# B&R Automation Studio project Ampel (part 6)

```cpp
	processRequest();
}

template <typename TG_, typename TA_>
HFSM2_CONSTEXPR(14)
void
R_<TG_, TA_>::immediateRestart(const StateID stateId_) noexcept {
	restart(stateId_);

	processRequest();
}

template <typename TG_, typename TA_>
HFSM2_CONSTEXPR(14)
void
R_<TG_, TA_>::immediateResume(const StateID stateId_) noexcept {
	resume(stateId_);

	processRequest();
}

template <typename TG_, typename TA_>
HFSM2_CONSTEXPR(14)
void
R_<TG_, TA_>::immediateSelect(const StateID stateId_) noexcept {
	select(stateId_);

	processRequest();
}

#if HFSM2_UTILITY_THEORY_AVAILABLE()

template <typename TG_, typename TA_>
HFSM2_CONSTEXPR(14)
void
R_<TG_, TA_>::immediateUtilize(const StateID stateId_) noexcept {
	utilize(stateId_);

	processRequest();
}

template <typename TG_, typename TA_>
HFSM2_CONSTEXPR(14)
void
R_<TG_, TA_>::immediateRandomize(const StateID stateId_) noexcept {
	randomize(stateId_);

	processRequest();
}

#endif

template <typename TG_, typename TA_>
HFSM2_CONSTEXPR(14)
void
R_<TG_, TA_>::reset() noexcept {
	HFSM2_ASSERT(_core.registry.isActive());

TransitionSets currentTransitions;
PlanControl control{_core, currentTransitions};

	_apex.deepExit(control);

	HFSM2_IF_TRANSITION_HISTORY(_core.transitionTargets.clear());
	HFSM2_IF_TRANSITION_HISTORY(_core.previousTransitions.clear());

	_core.registry.clear();
	// TODO: clear _core.requests
	// TODO: clear _core.rng			// HFSM2_IF_UTILITY_THEORY()
	// TODO: clear _core.planData		// HFSM2_IF_PLANS()
	// TODO: clear _activityHistory		// HFSM2_IF_STRUCTURE_REPORT()

_apex.deepRequestChange(control, {TransitionType::RESTART, INVALID_SHORT});
	_apex.deepEnter(control);
}

#if HFSM2_TRANSITION_HISTORY_AVAILABLE()

template <typename TG_, typename TA_>
HFSM2_CONSTEXPR(14)
bool
R_<TG_, TA_>::replayTransitions(const Transition* const transitions,
							  const Short count) noexcept
{
	HFSM2_ASSERT(transitions);
	HFSM2_ASSERT(_core.registry.isActive());

	_core.transitionTargets  .clear();
	_core.previousTransitions.clear();

	if (HFSM2_CHECKED(transitions && count)) {
TransitionSets currentTransitions;
PlanControl control{_core, currentTransitions};

		if (HFSM2_CHECKED(applyRequests(control, transitions, count))) {
for (Short i = 0; i < count; ++i)
				_core.previousTransitions.emplace(transitions[i]);

			_apex.deepChangeToRequested(control);

			_core.registry.clearRequests();

			HFSM2_IF_ASSERT(HFSM2_IF_PLANS(_core.planData.verifyPlans()));
			HFSM2_IF_STRUCTURE_REPORT(udpateActivity());

			return true;
		}
	}

	return false;
}

template <typename TG_, typename TA_>
template <Long NCount>
HFSM2_CONSTEXPR(14)
bool
R_<TG_, TA_>::replayTransitions(const DynamicArrayT<Transition, NCount>& transitions) noexcept {
	if (transitions.count())
		return replayTransitions(&transitions[0],
								 transitions.count());
	else
		return false;
}

template <typename TG_, typename TA_>
HFSM2_CONSTEXPR(14)
const typename R_<TG_, TA_>::Transition*
R_<TG_, TA_>::lastTransitionTo(const StateID stateId_) const noexcept {
	HFSM2_ASSERT(_core.registry.isActive());

	if (HFSM2_CHECKED(stateId_ < StateList::SIZE)) {
		const Short index = _core.transitionTargets[stateId_];

		if (index < _core.previousTransitions.count())
			return &_core.previousTransitions[index];
	}

	return nullptr;
}

#endif

template <typename TG_, typename TA_>
HFSM2_CONSTEXPR(14)
void
R_<TG_, TA_>::initialEnter() noexcept {
	HFSM2_ASSERT(!_core.registry.isActive());
	HFSM2_ASSERT(_core.requests.count() == 0);
	HFSM2_IF_TRANSITION_HISTORY(_core.transitionTargets.clear());
	HFSM2_IF_TRANSITION_HISTORY(HFSM2_ASSERT(_core.previousTransitions.count() == 0));

TransitionSets currentTransitions;
TransitionSet  pendingTransitions;

RegistryBackUp undo;
PlanControl control{_core, currentTransitions};

_apex.deepRequestChange(control, {TransitionType::RESTART, INVALID_SHORT});

	cancelledByEntryGuards(currentTransitions,
						   pendingTransitions);

for (Long i = 0;
		 i < SUBSTITUTION_LIMIT && _core.requests.count();
		 ++i)
	{
		backup(_core.registry, undo);

		if (applyRequests(currentTransitions,
						  control))
		{
pendingTransitions = _core.requests;
			_core.requests.clear();

			if (cancelledByEntryGuards(currentTransitions,
									   pendingTransitions))
			{
				HFSM2_BREAK();

				restore(_core.registry, undo);
			} else
currentTransitions += pendingTransitions;

			pendingTransitions.clear();
		} else
			_core.requests.clear();
	}
	HFSM2_ASSERT(_core.requests.count() == 0);
	HFSM2_IF_TRANSITION_HISTORY(_core.previousTransitions = currentTransitions);

	_apex.deepEnter(control);

	_core.registry.clearRequests();

	HFSM2_IF_ASSERT(HFSM2_IF_PLANS(_core.planData.verifyPlans()));
	HFSM2_IF_STRUCTURE_REPORT(udpateActivity());
}

template <typename TG_, typename TA_>
HFSM2_CONSTEXPR(14)
void
R_<TG_, TA_>::finalExit() noexcept {
	HFSM2_ASSERT(_core.registry.isActive());

TransitionSets emptyTransitions;
PlanControl control{_core, emptyTransitions};

	_apex.deepExit(control);

	_core.registry.clear();
	_core.requests.clear();

#if HFSM2_PLANS_AVAILABLE()
	_core.planData.clear();
#endif

#if HFSM2_UTILITY_THEORY_AVAILABLE()
	// TODO: _core.rng.clear();
#endif

#if HFSM2_TRANSITION_HISTORY_AVAILABLE()
	_core.transitionTargets  .clear();
	_core.previousTransitions.clear();
#endif

	HFSM2_IF_STRUCTURE_REPORT(udpateActivity());
}

template <typename TG_, typename TA_>
HFSM2_CONSTEXPR(14)
void
R_<TG_, TA_>::processRequest() noexcept {
	HFSM2_IF_ASSERT(HFSM2_IF_PLANS(_core.planData.verifyPlans()));

TransitionSets currentTransitions;
	HFSM2_IF_TRANSITION_HISTORY(_core.transitionTargets.clear());

	if (_core.requests.count()) {
		processTransitions(currentTransitions);

		HFSM2_IF_ASSERT(HFSM2_IF_PLANS(_core.planData.verifyPlans()));
		HFSM2_IF_STRUCTURE_REPORT(udpateActivity());
	}

	HFSM2_IF_TRANSITION_HISTORY(_core.previousTransitions = currentTransitions);
}

template <typename TG_, typename TA_>
HFSM2_CONSTEXPR(14)
void
R_<TG_, TA_>::processTransitions(TransitionSets& currentTransitions) noexcept {
	HFSM2_ASSERT(_core.registry.isActive());
	HFSM2_ASSERT(_core.requests.count());

TransitionSet pendingTransitions;

RegistryBackUp registryUndo;
PlanControl control{_core, currentTransitions};

for (Long i = 0;
		 i < SUBSTITUTION_LIMIT && _core.requests.count();
		 ++i)
	{
		backup(_core.registry, registryUndo);

		if (applyRequests(currentTransitions,
						  control))
		{
pendingTransitions = _core.requests;
			_core.requests.clear();

			if (cancelledByGuards(currentTransitions,
								  pendingTransitions))
			{
				HFSM2_IF_TRANSITION_HISTORY(_core.transitionTargets.clear());
				restore(_core.registry, registryUndo);
			} else
currentTransitions += pendingTransitions;

			pendingTransitions.clear();
		} else
			_core.requests.clear();
	}
	HFSM2_ASSERT(_core.requests.count() == 0);

	if (currentTransitions.count())
		_apex.deepChangeToRequested(control);

	_core.registry.clearRequests();
}

template <typename TG_, typename TA_>
HFSM2_CONSTEXPR(14)
bool
R_<TG_, TA_>::applyRequests(const TransitionSets& currentTransitions,
							Control& control) noexcept
{
bool changesMade = false;

for (Short i = 0; i < _core.requests.count(); ++i)
		changesMade |= applyRequest(currentTransitions, control, _core.requests[i], i);

return changesMade;
}

template <typename TG_, typename TA_>
HFSM2_CONSTEXPR(14)
bool
R_<TG_, TA_>::applyRequest(const TransitionSets& currentTransitions,
						   Control& control,
						   const Transition& request,
						   const Short index) noexcept
{
for (Short i = 0; i < currentTransitions.count(); ++i)
if (currentTransitions[i] == request)
			return false;

	switch (request.type) {
	case TransitionType::CHANGE:
	case TransitionType::RESTART:
	case TransitionType::RESUME:
	case TransitionType::SELECT:

#if HFSM2_UTILITY_THEORY_AVAILABLE()
	case TransitionType::UTILIZE:
	case TransitionType::RANDOMIZE:
#endif

		// TODO: have both return success status
		if (_core.registry.requestImmediate(request))
_apex.deepForwardActive(control, {request.type, index});
		else
_apex.deepRequest	   (control, {request.type, index});

		return true;

	case TransitionType::SCHEDULE:
		_core.registry.requestScheduled(request.destination);

		return false;

	default:
		HFSM2_BREAK();

		return false;
	}
}

template <typename TG_, typename TA_>
HFSM2_CONSTEXPR(14)
bool
R_<TG_, TA_>::cancelledByEntryGuards(const TransitionSets& currentTransitions,
									 const TransitionSet&  pendingTransitions) noexcept
{
GuardControl guardControl{_core,
							  currentTransitions,
							  pendingTransitions};

	return _apex.deepEntryGuard(guardControl);
}

template <typename TG_, typename TA_>
HFSM2_CONSTEXPR(14)
bool
R_<TG_, TA_>::cancelledByGuards(const TransitionSets& currentTransitions,
								const TransitionSet&  pendingTransitions) noexcept
{
GuardControl guardControl{_core,
							  currentTransitions,
							  pendingTransitions};

	return _apex.deepForwardExitGuard(guardControl) ||
		   _apex.deepForwardEntryGuard(guardControl);
}

#if HFSM2_SERIALIZATION_AVAILABLE()

template <typename TG_, typename TA_>
HFSM2_CONSTEXPR(14)
void
R_<TG_, TA_>::save(WriteStream& stream) const noexcept {
	HFSM2_ASSERT(_core.registry.isActive());

	_apex.deepSaveActive(_core.registry, stream);

	// TODO: save(stream, _core.requests);

#if HFSM2_PLANS_AVAILABLE()
	// TODO: save(stream, _core.planData);
#endif

#if HFSM2_UTILITY_THEORY_AVAILABLE()
	// TODO: save(stream, _core.rng);
#endif

#if HFSM2_TRANSITION_HISTORY_AVAILABLE()
	// TODO: save(stream, _core.transitionTargets);
	// TODO: save(stream, _core.previousTransitions);
#endif

#if HFSM2_STRUCTURE_REPORT_AVAILABLE()
	// TODO: save(stream, _activityHistory);
#endif
}

template <typename TG_, typename TA_>
HFSM2_CONSTEXPR(14)
void
R_<TG_, TA_>::load(ReadStream& stream) noexcept {
	HFSM2_ASSERT(_core.registry.isActive());

	_core.registry.clearRequests();
	_core.registry.compoResumable.clear();
	_apex.deepLoadRequested(_core.registry, stream);

	_core.requests.clear();
	// TODO: load(stream, _core.requests);

#if HFSM2_PLANS_AVAILABLE()
	_core.planData.clear();
	// TODO: load(stream, _core.planData);
#endif

#if HFSM2_UTILITY_THEORY_AVAILABLE()
	// TODO: load(stream, _core.rng);
#endif

#if HFSM2_TRANSITION_HISTORY_AVAILABLE()
	_core.transitionTargets  .clear();
	_core.previousTransitions.clear();
#endif

#if HFSM2_STRUCTURE_REPORT_AVAILABLE()
	// TODO: load(stream, _activityHistory);
#endif

TransitionSets emptyTransitions;
PlanControl control{_core, emptyTransitions};

	_apex.deepChangeToRequested(control);

	HFSM2_IF_STRUCTURE_REPORT(udpateActivity());
}

#endif

#if HFSM2_TRANSITION_HISTORY_AVAILABLE()

template <typename TG_, typename TA_>
HFSM2_CONSTEXPR(14)
bool
R_<TG_, TA_>::applyRequests(Control& control,
							const Transition* const transitions,
							const Short count) noexcept
{
TransitionSets currentTransitions;

	if (HFSM2_CHECKED(transitions && count)) {
bool changesMade = false;

for (Short i = 0; i < count; ++i)
			changesMade |= applyRequest(currentTransitions, control, transitions[i], i);

return changesMade;
	} else
		return false;
}

#endif

#if HFSM2_STRUCTURE_REPORT_AVAILABLE()

template <typename TG_, typename TA_>
HFSM2_CONSTEXPR(14)
void
R_<TG_, TA_>::getStateNames() noexcept {
StructureStateInfos stateInfos;
	_apex.deepGetNames(static_cast<Long>(-1), RegionType::COMPOSITE, 0, stateInfos);

Long margin = static_cast<Long>(-1);
for (Long s = 0; s < stateInfos.count(); ++s) {
const StructureStateInfo& stateInfo = stateInfos[s];
Prefix& prefix = _prefixes[s];

if (stateInfo.name[0] != '\0')
			_namedStates.set(s);

if (margin > stateInfo.depth && stateInfo.name[0] != '\0')
margin = stateInfo.depth;

		if (stateInfo.depth == 0)
prefix[0] = L'\0';
		else {
const Long mark = stateInfo.depth * 2 - 1;

prefix[mark + 0] = stateInfo.regionType == RegionType::COMPOSITE ? L'+' : L'+';
prefix[mark + 1] = L' ';
prefix[mark + 2] = L'\0';

for (Long d = mark; d > 0; --d)
prefix[d - 1] = L' ';

for (Long r = s; r > stateInfo.parent; --r) {
Prefix& prefixAbove = _prefixes[r - 1];

switch (prefixAbove[mark]) {
				case L' ':
prefixAbove[mark] = stateInfo.regionType == RegionType::COMPOSITE ? L'¦' : L'¦';
					break;
				case L'+':
prefixAbove[mark] = L'+';
					break;
				case L'+':
prefixAbove[mark] = L'¦';
					break;
				}
			}
		}
	}
	if (margin > 0)
		margin -= 1;

	_structure.clear();
for (Long s = 0; s < stateInfos.count(); ++s) {
const StructureStateInfo& stateInfo = stateInfos[s];
Prefix& prefix = _prefixes[s];
const Long space = stateInfo.depth * 2;

if (stateInfo.name[0] != L'\0') {
_structure.emplace(StructureEntry{false, &prefix[margin * 2], stateInfo.name});
			_activityHistory.emplace(static_cast<int8_t>(0));
		} else if (s + 1 < stateInfos.count()) {
Prefix& nextPrefix = _prefixes[s + 1];

			if (s > 0)
for (Long c = 0; c <= space; ++c)
nextPrefix[c] = prefix[c];

const Long mark = space + 1;

switch (nextPrefix[mark]) {
			case L'+':
nextPrefix[mark] = stateInfo.depth == margin ? L'+' : L'-';
				break;
			case L'¦':
nextPrefix[mark] = stateInfo.depth == margin ? L'+' : L'-';
				break;
			}
		}
	}
}

template <typename TG_, typename TA_>
HFSM2_CONSTEXPR(14)
void
R_<TG_, TA_>::udpateActivity() noexcept {
for (Long s = 0, i = 0; s < STATE_COUNT; ++s)
		if (_namedStates.get(s)) {
_structure[i].isActive = isActive(s);

typename ActivityHistory::Item& activity = _activityHistory[i];

if (_structure[i].isActive) {
				if (activity < 0)
activity = +1;
				else
activity = activity < INT8_MAX ? activity + 1 : activity;
			} else {
				if (activity > 0)
activity = -1;
				else
activity = activity > INT8_MIN ? activity - 1 : activity;
			}

++i;
		}
}

#endif

}
}

namespace hfsm2 {
	namespace detail {

		// Automatic / manual [de]activation

		template <
		typename
		, typename
		>
		class RV_;

		// Automatic enter() / exit()

		template <
		FeatureTag NFeatureTag
		, typename TContext
		, typename TReactOrder

#if HFSM2_UTILITY_THEORY_AVAILABLE()
		, typename TRank
		, typename TUtility
		, typename TRNG
#endif

		, Short NSubstitutionLimit
		HFSM2_IF_PLANS(, Long NTaskCapacity)
		, typename TPayload
		, typename TApex
		>
		class HFSM2_EMPTY_BASES RV_<
		G_<
		NFeatureTag
		, TContext
		, Automatic
		, TReactOrder
		HFSM2_IF_UTILITY_THEORY(, TRank, TUtility, TRNG)
		, NSubstitutionLimit
		HFSM2_IF_PLANS(, NTaskCapacity)
		, TPayload
		>
		, TApex
		>
		: public			R_ <
		G_<
		NFeatureTag
		, TContext
		, Automatic
		, TReactOrder
		HFSM2_IF_UTILITY_THEORY(, TRank, TUtility, TRNG)
		, NSubstitutionLimit
		HFSM2_IF_PLANS(, NTaskCapacity)
		, TPayload
		>
		, TApex
		>
		{
		using Base =		R_ <
			G_<
			NFeatureTag
			, TContext
			, Automatic
			, TReactOrder
		HFSM2_IF_UTILITY_THEORY(, TRank, TUtility, TRNG)
		, NSubstitutionLimit
		HFSM2_IF_PLANS(, NTaskCapacity)
		, TPayload
		>
		, TApex
		>;

		protected:
		using typename Base::Context;
		using typename Base::PureContext;

#if HFSM2_UTILITY_THEORY_AVAILABLE()
		using typename Base::RNG;
#endif

#if HFSM2_SERIALIZATION_AVAILABLE()
		using typename Base::Args;
		using typename Base::WriteStream;
		using typename Base::ReadStream;
#endif

#if HFSM2_LOG_INTERFACE_AVAILABLE()
		using typename Base::Logger;
#endif

		public:
		HFSM2_CONSTEXPR(14)	explicit RV_(Context& context
		HFSM2_IF_UTILITY_THEORY(, RNG& rng)
		HFSM2_IF_LOG_INTERFACE(, Logger* const logger = nullptr))	noexcept;

		HFSM2_CONSTEXPR(14)	explicit RV_(PureContext&& context
		HFSM2_IF_UTILITY_THEORY(, RNG& rng)
		HFSM2_IF_LOG_INTERFACE(, Logger* const logger = nullptr))	noexcept;

		HFSM2_CONSTEXPR(14)	RV_(const RV_&  other)													noexcept;
		HFSM2_CONSTEXPR(14)	RV_(	  RV_&& other)													noexcept;

		HFSM2_CONSTEXPR(20)	~RV_()																	noexcept;

#if HFSM2_SERIALIZATION_AVAILABLE()

		/// @brief Buffer for serialization
		/// @see `HFSM2_ENABLE_SERIALIZATION`
		using SerialBuffer			= typename Args::SerialBuffer;

		/// @brief Serialize FSM into 'buffer'
		/// @param buffer `SerialBuffer` to serialize to
		/// @see `HFSM2_ENABLE_SERIALIZATION`
		HFSM2_CONSTEXPR(14)	void save(		SerialBuffer& buffer)							  const noexcept;

		/// @brief De-serialize FSM from 'buffer'
		/// @param buffer `SerialBuffer` to de-serialize from
		/// @see `HFSM2_ENABLE_SERIALIZATION`
		HFSM2_CONSTEXPR(14)	void load(const SerialBuffer& buffer)									noexcept;

#endif

		private:
#if HFSM2_SERIALIZATION_AVAILABLE()
		using Base::save;
		using Base::load;
#endif

		private:
		using Base::initialEnter;
		using Base::finalExit;
	};

	// Manual enter() / exit()

	template <
	FeatureTag NFeatureTag
	, typename TContext
	, typename TReactOrder

#if HFSM2_UTILITY_THEORY_AVAILABLE()
	, typename TRank
	, typename TUtility
	, typename TRNG
#endif

	, Short NSubstitutionLimit
	HFSM2_IF_PLANS(, Long NTaskCapacity)
	, typename TPayload
	, typename TApex
	>
	class HFSM2_EMPTY_BASES RV_<
	G_<
	NFeatureTag
	, TContext
	, Manual
	, TReactOrder
	HFSM2_IF_UTILITY_THEORY(, TRank, TUtility, TRNG)
	, NSubstitutionLimit
	HFSM2_IF_PLANS(, NTaskCapacity)
	, TPayload
	>
	, TApex
	>
	: public			R_<
	G_<
	NFeatureTag
	, TContext
	, Manual
	, TReactOrder
	HFSM2_IF_UTILITY_THEORY(, TRank, TUtility, TRNG)
	, NSubstitutionLimit
	HFSM2_IF_PLANS(, NTaskCapacity)
	, TPayload
	>
	, TApex
	>
	{
	using Base =		R_<
		G_<
		NFeatureTag
		, TContext
		, Manual
		, TReactOrder
	HFSM2_IF_UTILITY_THEORY(, TRank, TUtility, TRNG)
	, NSubstitutionLimit
	HFSM2_IF_PLANS(, NTaskCapacity)
	, TPayload
	>
	, TApex
	>;

	public:
	using typename Base::Transition;

	protected:
#if HFSM2_UTILITY_THEORY_AVAILABLE()
	using typename Base::RNG;
#endif

#if HFSM2_SERIALIZATION_AVAILABLE()
	using typename Base::Args;
	using typename Base::WriteStream;
	using typename Base::ReadStream;
#endif

#if HFSM2_SERIALIZATION_AVAILABLE() || HFSM2_TRANSITION_HISTORY_AVAILABLE()
	using typename Base::PlanControl;
	using typename Base::TransitionSets;
#endif

	public:
	using Base::Base;

	/// @brief Check if FSM is active
	/// @return FSM active status
	HFSM2_CONSTEXPR(11)	bool isActive()													  const noexcept	{ return _core.registry.isActive();			}

	using Base::isActive;

	/// @brief Manually start the FSM
	///	  Can be used with UE4 to start / stop the FSM in `BeginPlay()` / `EndPlay()`
HFSM2_CONSTEXPR(14)	void enter()															noexcept	{ initialEnter(					);			}

	/// @brief Manually stop the FSM
	///   Can be used with UE4 to start / stop the FSM in `BeginPlay()` / `EndPlay()`
	HFSM2_CONSTEXPR(14)	void exit()																noexcept	{ finalExit();								}

#if HFSM2_SERIALIZATION_AVAILABLE()

	/// @brief Buffer for serialization
	/// @see `HFSM2_ENABLE_SERIALIZATION`
	using SerialBuffer			= typename Args::SerialBuffer;

	/// @brief Serialize FSM into 'buffer'
	/// @param buffer `SerialBuffer` to serialize to
	/// @see `HFSM2_ENABLE_SERIALIZATION`
	HFSM2_CONSTEXPR(14)	void save(		SerialBuffer& buffer)							  const noexcept;

	/// @brief De-serialize FSM from 'buffer'
	/// @param buffer `SerialBuffer` to de-serialize from
	/// @see `HFSM2_ENABLE_SERIALIZATION`
	HFSM2_CONSTEXPR(14)	void load(const SerialBuffer& buffer)									noexcept;

#endif

#if HFSM2_TRANSITION_HISTORY_AVAILABLE()

	/// @brief Start the FSM from a specific state
	///   Can be used to synchronize multiple FSMs
	/// @param `transitions` Array of 'Transition's to replay
	/// @param `count` Number of transitions
	/// @see `HFSM2_ENABLE_TRANSITION_HISTORY`
	HFSM2_CONSTEXPR(14)	bool replayEnter(const Transition* const transitions,
										 const Short count)										noexcept;

	/// @brief Start the FSM from a specific state
	///   Can be used to synchronize multiple FSMs
	/// @param `transitions` Array of 'Transition's to replay
	/// @see `HFSM2_ENABLE_TRANSITION_HISTORY`
	template <Long NCount>
	HFSM2_CONSTEXPR(14)	bool replayEnter(const DynamicArrayT<Transition, NCount>& transitions)	noexcept;

	/// @brief Start the FSM from a specific state
	///   Can be used to synchronize multiple FSMs
	/// @param `transition` 'Transition' to replay
	/// @see `HFSM2_ENABLE_TRANSITION_HISTORY`
	HFSM2_CONSTEXPR(14)	bool replayEnter(const Transition& transition)							noexcept	{ return replayEnter(&transition, 1);	}

#endif

private:
#if HFSM2_SERIALIZATION_AVAILABLE()
	using Base::save;
using Base::load;

	HFSM2_CONSTEXPR(14)	void loadEnter(ReadStream& stream)										noexcept;
#endif

protected:
	using Base::initialEnter;
using Base::finalExit;

using Base::_core;

#if HFSM2_SERIALIZATION_AVAILABLE() || HFSM2_TRANSITION_HISTORY_AVAILABLE()
	using Base::_apex;
#endif

#if HFSM2_TRANSITION_HISTORY_AVAILABLE()
	using Base::applyRequests;
	HFSM2_IF_STRUCTURE_REPORT(using Base::udpateActivity);
#endif
};

}
}

namespace hfsm2 {
	namespace detail {

		template <FeatureTag NFT_, typename TC_, typename TRO_ HFSM2_IF_UTILITY_THEORY(, typename TR_, typename TU_, typename TG_), Short NSL_ HFSM2_IF_PLANS(, Long NTC_), typename TP_, typename TA_>
		HFSM2_CONSTEXPR(14)
		RV_<G_<NFT_, TC_, Automatic, TRO_ HFSM2_IF_UTILITY_THEORY(, TR_, TU_, TG_), NSL_ HFSM2_IF_PLANS(, NTC_), TP_>, TA_>::RV_(Context& context
		HFSM2_IF_UTILITY_THEORY(, RNG& rng)
		HFSM2_IF_LOG_INTERFACE(, Logger* const logger)) noexcept
		: Base{context
		HFSM2_IF_UTILITY_THEORY(, rng)
	HFSM2_IF_LOG_INTERFACE(, logger)}
	{
	initialEnter();
}

template <FeatureTag NFT_, typename TC_, typename TRO_ HFSM2_IF_UTILITY_THEORY(, typename TR_, typename TU_, typename TG_), Short NSL_ HFSM2_IF_PLANS(, Long NTC_), typename TP_, typename TA_>
HFSM2_CONSTEXPR(14)
RV_<G_<NFT_, TC_, Automatic, TRO_ HFSM2_IF_UTILITY_THEORY(, TR_, TU_, TG_), NSL_ HFSM2_IF_PLANS(, NTC_), TP_>, TA_>::RV_(PureContext&& context
																													   HFSM2_IF_UTILITY_THEORY(, RNG& rng)
																													   HFSM2_IF_LOG_INTERFACE(, Logger* const logger)) noexcept
	: Base{move(context)
		 HFSM2_IF_UTILITY_THEORY(, rng)
		 HFSM2_IF_LOG_INTERFACE(, logger)}
{
	initialEnter();
}

template <FeatureTag NFT_, typename TC_, typename TRO_ HFSM2_IF_UTILITY_THEORY(, typename TR_, typename TU_, typename TG_), Short NSL_ HFSM2_IF_PLANS(, Long NTC_), typename TP_, typename TA_>
HFSM2_CONSTEXPR(14)
RV_<G_<NFT_, TC_, Automatic, TRO_ HFSM2_IF_UTILITY_THEORY(, TR_, TU_, TG_), NSL_ HFSM2_IF_PLANS(, NTC_), TP_>, TA_>::RV_(const RV_& other) noexcept
	: Base{other}
{}

template <FeatureTag NFT_, typename TC_, typename TRO_ HFSM2_IF_UTILITY_THEORY(, typename TR_, typename TU_, typename TG_), Short NSL_ HFSM2_IF_PLANS(, Long NTC_), typename TP_, typename TA_>
HFSM2_CONSTEXPR(14)
RV_<G_<NFT_, TC_, Automatic, TRO_ HFSM2_IF_UTILITY_THEORY(, TR_, TU_, TG_), NSL_ HFSM2_IF_PLANS(, NTC_), TP_>, TA_>::RV_(RV_&& other) noexcept
	: Base{move(other)}
{}

template <FeatureTag NFT_, typename TC_, typename TRO_ HFSM2_IF_UTILITY_THEORY(, typename TR_, typename TU_, typename TG_), Short NSL_ HFSM2_IF_PLANS(, Long NTC_), typename TP_, typename TA_>
HFSM2_CONSTEXPR(20)
RV_<G_<NFT_, TC_, Automatic, TRO_ HFSM2_IF_UTILITY_THEORY(, TR_, TU_, TG_), NSL_ HFSM2_IF_PLANS(, NTC_), TP_>, TA_>::~RV_() noexcept {
	finalExit();
}

#if HFSM2_SERIALIZATION_AVAILABLE()

template <FeatureTag NFT_, typename TC_, typename TRO_ HFSM2_IF_UTILITY_THEORY(, typename TR_, typename TU_, typename TG_), Short NSL_ HFSM2_IF_PLANS(, Long NTC_), typename TP_, typename TA_>
HFSM2_CONSTEXPR(14)
void
RV_<G_<NFT_, TC_, Automatic, TRO_ HFSM2_IF_UTILITY_THEORY(, TR_, TU_, TG_), NSL_ HFSM2_IF_PLANS(, NTC_), TP_>, TA_>::save(SerialBuffer& buffer) const noexcept {
WriteStream stream{buffer};

	stream.template write<1>(1);
	save(stream);
}

template <FeatureTag NFT_, typename TC_, typename TRO_ HFSM2_IF_UTILITY_THEORY(, typename TR_, typename TU_, typename TG_), Short NSL_ HFSM2_IF_PLANS(, Long NTC_), typename TP_, typename TA_>
HFSM2_CONSTEXPR(14)
void
RV_<G_<NFT_, TC_, Automatic, TRO_ HFSM2_IF_UTILITY_THEORY(, TR_, TU_, TG_), NSL_ HFSM2_IF_PLANS(, NTC_), TP_>, TA_>::load(const SerialBuffer& buffer) noexcept {
ReadStream stream{buffer};

	if (HFSM2_CHECKED(stream.template read<1>()))
		Base::load(stream);
}

#endif

#if HFSM2_SERIALIZATION_AVAILABLE()

template <FeatureTag NFT_, typename TC_, typename TRO_ HFSM2_IF_UTILITY_THEORY(, typename TR_, typename TU_, typename TG_), Short NSL_ HFSM2_IF_PLANS(, Long NTC_), typename TP_, typename TA_>
HFSM2_CONSTEXPR(14)
void
RV_<G_<NFT_, TC_, Manual, TRO_ HFSM2_IF_UTILITY_THEORY(, TR_, TU_, TG_), NSL_ HFSM2_IF_PLANS(, NTC_), TP_>, TA_>::save(SerialBuffer& buffer) const noexcept {
WriteStream stream{buffer};

	if (isActive()) {
		stream.template write<1>(1);

		save(stream);
	}
	else
		stream.template write<1>(0);
}

template <FeatureTag NFT_, typename TC_, typename TRO_ HFSM2_IF_UTILITY_THEORY(, typename TR_, typename TU_, typename TG_), Short NSL_ HFSM2_IF_PLANS(, Long NTC_), typename TP_, typename TA_>
HFSM2_CONSTEXPR(14)
void
RV_<G_<NFT_, TC_, Manual, TRO_ HFSM2_IF_UTILITY_THEORY(, TR_, TU_, TG_), NSL_ HFSM2_IF_PLANS(, NTC_), TP_>, TA_>::load(const SerialBuffer& buffer) noexcept {
ReadStream stream{buffer};

	if (stream.template read<1>()) {
		if (isActive())
			Base::load(stream);
		else
			loadEnter (stream);
	}
	else
		if (isActive())
			finalExit();
}

#endif

#if HFSM2_TRANSITION_HISTORY_AVAILABLE()

template <FeatureTag NFT_, typename TC_, typename TRO_ HFSM2_IF_UTILITY_THEORY(, typename TR_, typename TU_, typename TG_), Short NSL_ HFSM2_IF_PLANS(, Long NTC_), typename TP_, typename TA_>
HFSM2_CONSTEXPR(14)
bool
RV_<G_<NFT_, TC_, Manual, TRO_ HFSM2_IF_UTILITY_THEORY(, TR_, TU_, TG_), NSL_ HFSM2_IF_PLANS(, NTC_), TP_>, TA_>::replayEnter(const Transition* const transitions,
																															  const Short count) noexcept
{
	HFSM2_ASSERT(!_core.registry.isActive());
	HFSM2_ASSERT(_core.requests.count() == 0);

	_core.transitionTargets.clear();
	HFSM2_ASSERT(_core.previousTransitions.count() == 0);

	if (HFSM2_CHECKED(transitions && count)) {
TransitionSets emptyTransitions;
PlanControl control{_core, emptyTransitions};

		if (HFSM2_CHECKED(applyRequests(control, transitions, count))) {
for (Short i = 0; i < count; ++i)
				_core.previousTransitions.emplace(transitions[i]);

			_apex.deepEnter(control);

			_core.registry.clearRequests();

			HFSM2_IF_ASSERT(HFSM2_IF_PLANS(_core.planData.verifyPlans()));
			HFSM2_IF_STRUCTURE_REPORT(udpateActivity());

			return true;
		}
	}

	return false;
}

template <FeatureTag NFT_, typename TC_, typename TRO_ HFSM2_IF_UTILITY_THEORY(, typename TR_, typename TU_, typename TG_), Short NSL_ HFSM2_IF_PLANS(, Long NTC_), typename TP_, typename TA_>
template <Long NCount>
HFSM2_CONSTEXPR(14)
bool
RV_<G_<NFT_, TC_, Manual, TRO_ HFSM2_IF_UTILITY_THEORY(, TR_, TU_, TG_), NSL_ HFSM2_IF_PLANS(, NTC_), TP_>, TA_>::replayEnter(const DynamicArrayT<Transition, NCount>& transitions)  noexcept {
	if (transitions.count())
		return replayEnter(&transitions[0],
						   transitions.count());
	else
		return false;
}

#endif

#if HFSM2_SERIALIZATION_AVAILABLE()

template <FeatureTag NFT_, typename TC_, typename TRO_ HFSM2_IF_UTILITY_THEORY(, typename TR_, typename TU_, typename TG_), Short NSL_ HFSM2_IF_PLANS(, Long NTC_), typename TP_, typename TA_>
HFSM2_CONSTEXPR(14)
void
RV_<G_<NFT_, TC_, Manual, TRO_ HFSM2_IF_UTILITY_THEORY(, TR_, TU_, TG_), NSL_ HFSM2_IF_PLANS(, NTC_), TP_>, TA_>::loadEnter(ReadStream& stream) noexcept {
	HFSM2_ASSERT(_core.registry.empty());
	_apex.deepLoadRequested(_core.registry, stream);

	HFSM2_ASSERT(_core.requests.empty());

#if HFSM2_PLANS_AVAILABLE()
	HFSM2_ASSERT(_core.planData.empty() == 0);
#endif

#if HFSM2_TRANSITION_HISTORY_AVAILABLE()
	HFSM2_ASSERT(_core.transitionTargets  .empty());
	HFSM2_ASSERT(_core.previousTransitions.empty());
#endif

#if HFSM2_STRUCTURE_REPORT_AVAILABLE()
	//HFSM2_ASSERT(_activityHistory.empty());
#endif

TransitionSets emptyTransitions;
PlanControl control{_core, emptyTransitions};

	_apex.deepEnter(control);

	HFSM2_IF_STRUCTURE_REPORT(udpateActivity());
}

#endif

}
}

namespace hfsm2 {
	namespace detail {

		template <
		typename
		, typename
		>
		class RP_;

		// Non-'void' payloads

		template <
		FeatureTag NFeatureTag
		, typename TContext
		, typename TActivation
		, typename TReactOrder

#if HFSM2_UTILITY_THEORY_AVAILABLE()
		, typename TRank
		, typename TUtility
		, typename TRNG
#endif

		, Short NSubstitutionLimit
		HFSM2_IF_PLANS(, Long NTaskCapacity)
		, typename TPayload
		, typename TApex
		>
		class HFSM2_EMPTY_BASES RP_<
		G_<
		NFeatureTag
		, TContext
		, TActivation
		, TReactOrder
		HFSM2_IF_UTILITY_THEORY(, TRank, TUtility, TRNG)
		, NSubstitutionLimit
		HFSM2_IF_PLANS(, NTaskCapacity)
		, TPayload
		>
		, TApex
		>
		: public			RV_<
		G_<
		NFeatureTag
		, TContext
		, TActivation
		, TReactOrder
		HFSM2_IF_UTILITY_THEORY(, TRank, TUtility, TRNG)
		, NSubstitutionLimit
		HFSM2_IF_PLANS(, NTaskCapacity)
		, TPayload
		>
		, TApex
		>
		{
		using Base =		RV_<
			G_<
			NFeatureTag
			, TContext
			, TActivation
			, TReactOrder
		HFSM2_IF_UTILITY_THEORY(, TRank, TUtility, TRNG)
		, NSubstitutionLimit
		HFSM2_IF_PLANS(, NTaskCapacity)
		, TPayload
		>
		, TApex
		>;

		using Transition			= TransitionT<TPayload>;

		public:
		using typename Base::Payload;

#if HFSM2_UTILITY_THEORY_AVAILABLE()
		using typename Base::RNG;
#endif

		public:
		using Base::Base;
		using Base::processRequest;

		/// @brief Get state identifier for a state type
		/// @tparam `TState` State type
		/// @return Numeric state identifier
		template <typename TState>
		static
	HFSM2_CONSTEXPR(11) StateID  stateId()											noexcept	{ return Base::template stateId<TState>();		}

	/// @brief Get region identifier for a region type
	/// @tparam `TState` Region head state type
	/// @return Numeric region identifier
	template <typename TState>
	static
HFSM2_CONSTEXPR(11) RegionID regionId()											noexcept	{ return Base::template regionId<TState>();		}

	/// @brief Queue a transition into a state (takes effect during `immediate*()`, `update()` or `react()`)
	///   (if transitioning into a region, acts depending on the region type)
	/// @param `stateId` Destination state identifier
	/// @param `payload` Payload
	HFSM2_CONSTEXPR(14)	void changeWith				(const StateID  stateId_,
													 const Payload& payload)		noexcept;

	/// @brief Queue a transition into a state (takes effect during `immediate*()`, `update()` or `react()`)
	///   (if transitioning into a region, acts depending on the region type)
	/// @tparam `TState` Destination state type
	/// @param `payload` Payload
	template <typename TState>
	HFSM2_CONSTEXPR(14)	void changeWith				(const Payload& payload)		noexcept	{ changeWith   (stateId<TState>(), payload );	}

	/// @brief Queue a transition into a state (takes effect during `immediate*()`, `update()` or `react()`)
	///   (if transitioning into a region, activates the initial state)
	/// @param `stateId` Destination state identifier
	/// @param `payload` Payload
	HFSM2_CONSTEXPR(14)	void restartWith			(const StateID  stateId_,
													 const Payload& payload)		noexcept;

	/// @brief Queue a transition into a state (takes effect during `immediate*()`, `update()` or `react()`)
	///   (if transitioning into a region, activates the initial state)
	/// @tparam `TState` Destination state type
	/// @param `payload` Payload
	template <typename TState>
	HFSM2_CONSTEXPR(14)	void restartWith			(const Payload& payload)		noexcept	{ restartWith  (stateId<TState>(), payload );	}

	/// @brief Queue a transition into a state (takes effect during `immediate*()`, `update()` or `react()`)
	///   (if transitioning into a region, activates the state that was active previously)
	/// @param `stateId` Destination state identifier
	/// @param `payload` Payload
	HFSM2_CONSTEXPR(14)	void resumeWith				(const StateID  stateId_,
													 const Payload& payload)		noexcept;

	/// @brief Queue a transition into a state (takes effect during `immediate*()`, `update()` or `react()`)
	///   (if transitioning into a region, activates the state that was active previously)
	/// @tparam `TState` Destination state type
	/// @param `payload` Payload
	template <typename TState>
	HFSM2_CONSTEXPR(14)	void resumeWith				(const Payload& payload)		noexcept	{ resumeWith   (stateId<TState>(), payload );	}

	/// @brief Queue a transition into a state (takes effect during `immediate*()`, `update()` or `react()`)
	///   (if transitioning into a region, activates the sub-state by index returned by the region's `select()` method)
	/// @param `stateId` Destination state identifier
	/// @param `payload` Payload
	HFSM2_CONSTEXPR(14)	void selectWith				(const StateID  stateId_,
													 const Payload& payload)		noexcept;

	/// @brief Queue a transition into a state (takes effect during `immediate*()`, `update()` or `react()`)
	///   (if transitioning into a region, activates the sub-state by index returned by the region's `select()` method)
	/// @tparam `TState` Destination state type
	/// @param `payload` Payload
	template <typename TState>
	HFSM2_CONSTEXPR(14)	void selectWith				(const Payload& payload)		noexcept	{ selectWith   (stateId<TState>(), payload );	}

#if HFSM2_UTILITY_THEORY_AVAILABLE()

	/// @brief Queue a transition into a state (takes effect during `immediate*()`, `update()` or `react()`)
	///   (if transitioning into a region, activates the state with the highest `utility()`
	///   among those with the highest `rank()`)
	/// @param `stateId` Destination state identifier
	/// @param `payload` Payload
	/// @see `HFSM2_ENABLE_UTILITY_THEORY`
	HFSM2_CONSTEXPR(14)	void utilizeWith			(const StateID  stateId_,
													 const Payload& payload)		noexcept;

	/// @brief Queue a transition into a state (takes effect during `immediate*()`, `update()` or `react()`)
	///   (if transitioning into a region, activates the state with the highest `utility()`
	///   among those with the highest `rank()`)
	/// @tparam `TState` Destination state type
	/// @param `payload` Payload
	/// @see `HFSM2_ENABLE_UTILITY_THEORY`
	template <typename TState>
	HFSM2_CONSTEXPR(14)	void utilizeWith			(const Payload& payload)		noexcept	{ utilizeWith  (stateId<TState>(), payload );	}

	/// @brief Queue a transition into a state (takes effect during `immediate*()`, `update()` or `react()`)
	///   (if transitioning into a region, uses weighted random to activate the state proportional to `utility()`
	///   among those with the highest `rank()`)
	/// @param `stateId` Destination state identifier
	/// @param `payload` Payload
	/// @see `HFSM2_ENABLE_UTILITY_THEORY`
	HFSM2_CONSTEXPR(14)	void randomizeWith			(const StateID  stateId_,
													 const Payload& payload)		noexcept;

	/// @brief Queue a transition into a state (takes effect during `immediate*()`, `update()` or `react()`)
	///   (if transitioning into a region, uses weighted random to activate the state proportional to `utility()`
	///   among those with the highest `rank()`)
	/// @tparam `TState` Destination state type
	/// @param `payload` Payload
	/// @see `HFSM2_ENABLE_UTILITY_THEORY`
	template <typename TState>
	HFSM2_CONSTEXPR(14)	void randomizeWith			(const Payload& payload)		noexcept	{ randomizeWith(stateId<TState>(), payload );	}

#endif

	/// @brief Schedule a state to be activated when its parent region is activated
	/// @param `stateId` Destination state identifier
	/// @param `payload` Payload
	HFSM2_CONSTEXPR(14)	void scheduleWith			(const StateID  stateId_,
													 const Payload& payload)		noexcept;

	/// @brief Schedule a state to be activated when its parent region is activated
	/// @tparam `TState` Destination state type
	/// @param `payload` Payload
	template <typename TState>
	HFSM2_CONSTEXPR(14)	void scheduleWith			(const Payload& payload)		noexcept	{ scheduleWith (stateId<TState>(), payload );	}

	/// @brief Transition into a state
	///   (if transitioning into a region, acts depending on the region type)
	/// @param `stateId` Destination state identifier
	/// @param `payload` Payload
	/// @see `changeWith()`
	HFSM2_CONSTEXPR(14)	void immediateChangeWith	(const StateID  stateId_,
													 const Payload& payload)		noexcept;

	/// @brief Transition into a state
	///   (if transitioning into a region, acts depending on the region type)
	/// @tparam `TState` Destination state type
	/// @param `payload` Payload
	/// @see `changeWith()`
	template <typename TState>
	HFSM2_CONSTEXPR(14)	void immediateChangeWith	(const Payload& payload)		noexcept	{ immediateChangeWith   (stateId<TState>(), payload );	}

	/// @brief Transition into a state (if transitioning into a region, activates the initial state)
	/// @param `stateId` Destination state identifier
	/// @param `payload` Payload
	/// @see `restartWith()`
	HFSM2_CONSTEXPR(14)	void immediateRestartWith	(const StateID  stateId_,
													 const Payload& payload)		noexcept;

	/// @brief Transition into a state (if transitioning into a region, activates the initial state)
	/// @tparam `TState` Destination state type
	/// @param `payload` Payload
	/// @see `restartWith()`
	template <typename TState>
	HFSM2_CONSTEXPR(14)	void immediateRestartWith	(const Payload& payload)		noexcept	{ immediateRestartWith	(stateId<TState>(), payload );	}

	/// @brief Transition into a state
	///   (if transitioning into a region, activates the state that was active previously)
	/// @param `stateId` Destination state identifier
	/// @param `payload` Payload
	/// @see `resumeWith()`
	HFSM2_CONSTEXPR(14)	void immediateResumeWith	(const StateID  stateId_,
													 const Payload& payload)		noexcept;

	/// @brief Transition into a state
	///   (if transitioning into a region, activates the state that was active previously)
	/// @tparam `TState` Destination state type
	/// @param `payload` Payload
	/// @see `resumeWith()`
	template <typename TState>
	HFSM2_CONSTEXPR(14)	void immediateResumeWith	(const Payload& payload)		noexcept	{ immediateResumeWith	(stateId<TState>(), payload );	}

	/// @brief Transition into a state
	///   (if transitioning into a region, activates the sub-state by index returned by the region's `select()` method)
	/// @param `stateId` Destination state identifier
	/// @param `payload` Payload
	/// @see `selectWith()`
	HFSM2_CONSTEXPR(14)	void immediateSelectWith	(const StateID  stateId_,
													 const Payload& payload)		noexcept;

	/// @brief Transition into a state
	///   (if transitioning into a region, activates the sub-state by index returned by the region's `select()` method)
	/// @tparam `TState` Destination state type
	/// @param `payload` Payload
	/// @see `selectWith()`
	template <typename TState>
	HFSM2_CONSTEXPR(14)	void immediateSelectWith	(const Payload& payload)		noexcept	{ immediateSelectWith	(stateId<TState>(), payload );	}

#if HFSM2_UTILITY_THEORY_AVAILABLE()

	/// @brief Transition into a state
	///   (if transitioning into a region, activates the state with the highest `utility()`
	///   among those with the highest `rank()`)
	/// @param `stateId` Destination state identifier
	/// @param `payload` Payload
	/// @see `utilizeWith()`
	/// @see `HFSM2_ENABLE_UTILITY_THEORY`
	HFSM2_CONSTEXPR(14)	void immediateUtilizeWith	(const StateID  stateId_,
													 const Payload& payload)		noexcept;

	/// @brief Transition into a state
	///   (if transitioning into a region, activates the state with the highest `utility()`
	///   among those with the highest `rank()`)
	/// @tparam `TState` Destination state type
	/// @param `payload` Payload
	/// @see `utilizeWith()`
	/// @see `HFSM2_ENABLE_UTILITY_THEORY`
	template <typename TState>
	HFSM2_CONSTEXPR(14)	void immediateUtilizeWith	(const Payload& payload)		noexcept	{ immediateUtilizeWith	(stateId<TState>(), payload );	}

	/// @brief Transition into a state
	///   (if transitioning into a region, uses weighted random to activate the state proportional to `utility()`
	///   among those with the highest `rank()`)
	/// @param `stateId` Destination state identifier
	/// @param `payload` Payload
	/// @see `randomizeWith()`
	/// @see `HFSM2_ENABLE_UTILITY_THEORY`
	HFSM2_CONSTEXPR(14)	void immediateRandomizeWith	(const StateID  stateId_,
													 const Payload& payload)		noexcept;

	/// @brief Transition into a state
	///   (if transitioning into a region, uses weighted random to activate the state proportional to `utility()`
	///   among those with the highest `rank()`)
	/// @tparam `TState` Destination state type
	/// @param `payload` Payload
	/// @see `randomizeWith()`
	/// @see `HFSM2_ENABLE_UTILITY_THEORY`
	template <typename TState>
	HFSM2_CONSTEXPR(14)	void immediateRandomizeWith	(const Payload& payload)		noexcept	{ immediateRandomizeWith(stateId<TState>(), payload );	}

#endif

protected:
	using Base::_core;
};

template <
	FeatureTag NFeatureTag
  , typename TContext
  , typename TActivation
  , typename TReactOrder

#if HFSM2_UTILITY_THEORY_AVAILABLE()
, typename TRank
, typename TUtility
  , typename TRNG
#endif

, Short NSubstitutionLimit
  HFSM2_IF_PLANS(, Long NTaskCapacity)
  , typename TApex
>
class HFSM2_EMPTY_BASES RP_<
							G_<
								NFeatureTag
							  , TContext
							  , TActivation
							  , TReactOrder
							  HFSM2_IF_UTILITY_THEORY(, TRank, TUtility, TRNG)
							  , NSubstitutionLimit
							  HFSM2_IF_PLANS(, NTaskCapacity)
							  , void
							>
						  , TApex
						>
	: public			RV_<
							G_<
								NFeatureTag
							  , TContext
							  , TActivation
							  , TReactOrder
							  HFSM2_IF_UTILITY_THEORY(, TRank, TUtility, TRNG)
							  , NSubstitutionLimit
							  HFSM2_IF_PLANS(, NTaskCapacity)
							  , void
							>
						  , TApex
						>
{
	using Base =		RV_<
	G_<
	NFeatureTag
	, TContext
	, TActivation
	, TReactOrder
							  HFSM2_IF_UTILITY_THEORY(, TRank, TUtility, TRNG)
							  , NSubstitutionLimit
							  HFSM2_IF_PLANS(, NTaskCapacity)
							  , void
							>
						  , TApex
						>;

public:
#if HFSM2_UTILITY_THEORY_AVAILABLE()
	using typename Base::RNG;
#endif

	using Base::Base;
};

}
}

namespace hfsm2 {
	namespace detail {

		template <FeatureTag NFT_, typename TC_, typename TV_, typename TRO_ HFSM2_IF_UTILITY_THEORY(, typename TR_, typename TU_, typename TG_), Short NSL_ HFSM2_IF_PLANS(, Long NTC_), typename TP_, typename TA_>
		HFSM2_CONSTEXPR(14)
		void
		RP_<G_<NFT_, TC_, TV_, TRO_ HFSM2_IF_UTILITY_THEORY(, TR_, TU_, TG_), NSL_ HFSM2_IF_PLANS(, NTC_), TP_>, TA_>::changeWith(const StateID  stateId_,
		const Payload& payload) noexcept
		{
		HFSM2_ASSERT(_core.registry.isActive());

		_core.requests.emplace(Transition{stateId_, TransitionType::CHANGE, payload});

		HFSM2_LOG_TRANSITION(_core.context, INVALID_STATE_ID, TransitionType::CHANGE, stateId_);
	}

	template <FeatureTag NFT_, typename TC_, typename TV_, typename TRO_ HFSM2_IF_UTILITY_THEORY(, typename TR_, typename TU_, typename TG_), Short NSL_ HFSM2_IF_PLANS(, Long NTC_), typename TP_, typename TA_>
	HFSM2_CONSTEXPR(14)
	void
	RP_<G_<NFT_, TC_, TV_, TRO_ HFSM2_IF_UTILITY_THEORY(, TR_, TU_, TG_), NSL_ HFSM2_IF_PLANS(, NTC_), TP_>, TA_>::restartWith(const StateID  stateId_,
	const Payload& payload) noexcept
	{
	HFSM2_ASSERT(_core.registry.isActive());

	_core.requests.emplace(Transition{stateId_, TransitionType::RESTART, payload});

	HFSM2_LOG_TRANSITION(_core.context, INVALID_STATE_ID, TransitionType::RESTART, stateId_);
}

template <FeatureTag NFT_, typename TC_, typename TV_, typename TRO_ HFSM2_IF_UTILITY_THEORY(, typename TR_, typename TU_, typename TG_), Short NSL_ HFSM2_IF_PLANS(, Long NTC_), typename TP_, typename TA_>
HFSM2_CONSTEXPR(14)
void
RP_<G_<NFT_, TC_, TV_, TRO_ HFSM2_IF_UTILITY_THEORY(, TR_, TU_, TG_), NSL_ HFSM2_IF_PLANS(, NTC_), TP_>, TA_>::resumeWith(const StateID  stateId_,
																														  const Payload& payload) noexcept
{
	HFSM2_ASSERT(_core.registry.isActive());

_core.requests.emplace(Transition{stateId_, TransitionType::RESUME, payload});

	HFSM2_LOG_TRANSITION(_core.context, INVALID_STATE_ID, TransitionType::RESUME, stateId_);
}

template <FeatureTag NFT_, typename TC_, typename TV_, typename TRO_ HFSM2_IF_UTILITY_THEORY(, typename TR_, typename TU_, typename TG_), Short NSL_ HFSM2_IF_PLANS(, Long NTC_), typename TP_, typename TA_>
HFSM2_CONSTEXPR(14)
void
RP_<G_<NFT_, TC_, TV_, TRO_ HFSM2_IF_UTILITY_THEORY(, TR_, TU_, TG_), NSL_ HFSM2_IF_PLANS(, NTC_), TP_>, TA_>::selectWith(const StateID  stateId_,
																														  const Payload& payload) noexcept
{
	HFSM2_ASSERT(_core.registry.isActive());

_core.requests.emplace(Transition{stateId_, TransitionType::SELECT, payload});

	HFSM2_LOG_TRANSITION(_core.context, INVALID_STATE_ID, TransitionType::SELECT, stateId_);
}

#if HFSM2_UTILITY_THEORY_AVAILABLE()

template <FeatureTag NFT_, typename TC_, typename TV_, typename TRO_, typename TR_, typename TU_, typename TG_, Short NSL_ HFSM2_IF_PLANS(, Long NTC_), typename TP_, typename TA_>
HFSM2_CONSTEXPR(14)
void
RP_<G_<NFT_, TC_, TV_, TRO_, TR_, TU_, TG_, NSL_ HFSM2_IF_PLANS(, NTC_), TP_>, TA_>::utilizeWith(const StateID  stateId_,
																								 const Payload& payload) noexcept
{
	HFSM2_ASSERT(_core.registry.isActive());

_core.requests.emplace(Transition{stateId_, TransitionType::UTILIZE, payload});

	HFSM2_LOG_TRANSITION(_core.context, INVALID_STATE_ID, TransitionType::UTILIZE, stateId_);
}

template <FeatureTag NFT_, typename TC_, typename TV_, typename TRO_, typename TR_, typename TU_, typename TG_, Short NSL_ HFSM2_IF_PLANS(, Long NTC_), typename TP_, typename TA_>
HFSM2_CONSTEXPR(14)
void
	RP_<G_<NFT_, TC_, TV_, TRO_, TR_, TU_, TG_, NSL_ HFSM2_IF_PLANS(, NTC_), TP_>, TA_>::randomizeWith(const StateID  stateId_,
																								   const Payload& payload) noexcept
{
	HFSM2_ASSERT(_core.registry.isActive());

_core.requests.emplace(Transition{stateId_, TransitionType::RANDOMIZE, payload});

	HFSM2_LOG_TRANSITION(_core.context, INVALID_STATE_ID, TransitionType::RANDOMIZE, stateId_);
}

#endif

template <FeatureTag NFT_, typename TC_, typename TV_, typename TRO_ HFSM2_IF_UTILITY_THEORY(, typename TR_, typename TU_, typename TG_), Short NSL_ HFSM2_IF_PLANS(, Long NTC_), typename TP_, typename TA_>
HFSM2_CONSTEXPR(14)
void
RP_<G_<NFT_, TC_, TV_, TRO_ HFSM2_IF_UTILITY_THEORY(, TR_, TU_, TG_), NSL_ HFSM2_IF_PLANS(, NTC_), TP_>, TA_>::scheduleWith(const StateID  stateId_,
																															const Payload& payload) noexcept
{
	HFSM2_ASSERT(_core.registry.isActive());

_core.requests.emplace(Transition{stateId_, TransitionType::SCHEDULE, payload});

	HFSM2_LOG_TRANSITION(_core.context, INVALID_STATE_ID, TransitionType::SCHEDULE, stateId_);
}

template <FeatureTag NFT_, typename TC_, typename TV_, typename TRO_ HFSM2_IF_UTILITY_THEORY(, typename TR_, typename TU_, typename TG_), Short NSL_ HFSM2_IF_PLANS(, Long NTC_), typename TP_, typename TA_>
HFSM2_CONSTEXPR(14)
void
RP_<G_<NFT_, TC_, TV_, TRO_ HFSM2_IF_UTILITY_THEORY(, TR_, TU_, TG_), NSL_ HFSM2_IF_PLANS(, NTC_), TP_>, TA_>::immediateChangeWith(const StateID  stateId_,
																																   const Payload& payload) noexcept
{
	changeWith(stateId_, payload);

	processRequest();
}

template <FeatureTag NFT_, typename TC_, typename TV_, typename TRO_ HFSM2_IF_UTILITY_THEORY(, typename TR_, typename TU_, typename TG_), Short NSL_ HFSM2_IF_PLANS(, Long NTC_), typename TP_, typename TA_>
HFSM2_CONSTEXPR(14)
void
RP_<G_<NFT_, TC_, TV_, TRO_ HFSM2_IF_UTILITY_THEORY(, TR_, TU_, TG_), NSL_ HFSM2_IF_PLANS(, NTC_), TP_>, TA_>::immediateRestartWith(const StateID  stateId_,
																																	const Payload& payload) noexcept
{
	restartWith(stateId_, payload);

	processRequest();
}

template <FeatureTag NFT_, typename TC_, typename TV_, typename TRO_ HFSM2_IF_UTILITY_THEORY(, typename TR_, typename TU_, typename TG_), Short NSL_ HFSM2_IF_PLANS(, Long NTC_), typename TP_, typename TA_>
HFSM2_CONSTEXPR(14)
void
RP_<G_<NFT_, TC_, TV_, TRO_ HFSM2_IF_UTILITY_THEORY(, TR_, TU_, TG_), NSL_ HFSM2_IF_PLANS(, NTC_), TP_>, TA_>::immediateResumeWith(const StateID  stateId_,
																																   const Payload& payload) noexcept
{
	resumeWith(stateId_, payload);

	processRequest();
}

template <FeatureTag NFT_, typename TC_, typename TV_, typename TRO_ HFSM2_IF_UTILITY_THEORY(, typename TR_, typename TU_, typename TG_), Short NSL_ HFSM2_IF_PLANS(, Long NTC_), typename TP_, typename TA_>
HFSM2_CONSTEXPR(14)
void
RP_<G_<NFT_, TC_, TV_, TRO_ HFSM2_IF_UTILITY_THEORY(, TR_, TU_, TG_), NSL_ HFSM2_IF_PLANS(, NTC_), TP_>, TA_>::immediateSelectWith(const StateID  stateId_,
																																   const Payload& payload) noexcept
{
	selectWith(stateId_, payload);

	processRequest();
}

#if HFSM2_UTILITY_THEORY_AVAILABLE()

template <FeatureTag NFT_, typename TC_, typename TV_, typename TRO_, typename TR_, typename TU_, typename TG_, Short NSL_ HFSM2_IF_PLANS(, Long NTC_), typename TP_, typename TA_>
HFSM2_CONSTEXPR(14)
void
	RP_<G_<NFT_, TC_, TV_, TRO_, TR_, TU_, TG_, NSL_ HFSM2_IF_PLANS(, NTC_), TP_>, TA_>::immediateUtilizeWith(const StateID  stateId_,
																										  const Payload& payload) noexcept
{
	utilizeWith(stateId_, payload);

	processRequest();
}

template <FeatureTag NFT_, typename TC_, typename TV_, typename TRO_, typename TR_, typename TU_, typename TG_, Short NSL_ HFSM2_IF_PLANS(, Long NTC_), typename TP_, typename TA_>
HFSM2_CONSTEXPR(14)
void
	RP_<G_<NFT_, TC_, TV_, TRO_, TR_, TU_, TG_, NSL_ HFSM2_IF_PLANS(, NTC_), TP_>, TA_>::immediateRandomizeWith(const StateID  stateId_,
																											const Payload& payload) noexcept
{
	randomizeWith(stateId_, payload);

	processRequest();
}

#endif

}
}

namespace hfsm2 {
	namespace detail {

		template <
		typename
		, typename
		>
		class RC_;

		// TContext

		template <
		FeatureTag NFeatureTag
		, typename TContext
		, typename TActivation
		, typename TReactOrder

#if HFSM2_UTILITY_THEORY_AVAILABLE()
		, typename TRank
		, typename TUtility
		, typename TRNG
#endif

		, Short NSubstitutionLimit
		HFSM2_IF_PLANS(, Long NTaskCapacity)
		, typename TPayload
		, typename TApex
		>
		class HFSM2_EMPTY_BASES RC_<
		G_<
		NFeatureTag
		, TContext
		, TActivation
		, TReactOrder
		HFSM2_IF_UTILITY_THEORY(, TRank, TUtility, TRNG)
		, NSubstitutionLimit
		HFSM2_IF_PLANS(, NTaskCapacity)
		, TPayload
		>
		, TApex
		>
		: public			RP_<
		G_<
		NFeatureTag
		, TContext
		, TActivation
		, TReactOrder
		HFSM2_IF_UTILITY_THEORY(, TRank, TUtility, TRNG)
		, NSubstitutionLimit
		HFSM2_IF_PLANS(, NTaskCapacity)
		, TPayload
		>
		, TApex
		>
		{
		using Base =		RP_<
			G_<
			NFeatureTag
			, TContext
			, TActivation
			, TReactOrder
		HFSM2_IF_UTILITY_THEORY(, TRank, TUtility, TRNG)
		, NSubstitutionLimit
		HFSM2_IF_PLANS(, NTaskCapacity)
		, TPayload
		>
		, TApex
		>;

		public:
		static constexpr FeatureTag FEATURE_TAG = Base::FEATURE_TAG;

		using typename Base::Context;
		using typename Base::PureContext;

#if HFSM2_UTILITY_THEORY_AVAILABLE()
		using typename Base::RNG;
#endif

#if HFSM2_LOG_INTERFACE_AVAILABLE()
		using typename Base::Logger;
#endif

		public:
		HFSM2_CONSTEXPR(14)	explicit RC_(Context& context
		HFSM2_IF_UTILITY_THEORY(, RNG& rng)
		HFSM2_IF_LOG_INTERFACE(, Logger* const logger = nullptr))	noexcept;

		HFSM2_CONSTEXPR(14)	explicit RC_(PureContext&& context
		HFSM2_IF_UTILITY_THEORY(, RNG& rng)
		HFSM2_IF_LOG_INTERFACE(, Logger* const logger = nullptr))	noexcept;

		HFSM2_CONSTEXPR(NO) RC_(const RC_& )														noexcept = default;
		HFSM2_CONSTEXPR(NO) RC_(	  RC_&&)														noexcept = default;

		private:
		using Base::_core;
	};

	// TContext&

	template <
	FeatureTag NFeatureTag
	, typename TContext
	, typename TActivation
	, typename TReactOrder

#if HFSM2_UTILITY_THEORY_AVAILABLE()
	, typename TRank
	, typename TUtility
	, typename TRNG
#endif

	, Short NSubstitutionLimit
	HFSM2_IF_PLANS(, Long NTaskCapacity)
	, typename TPayload
	, typename TApex
	>
	class HFSM2_EMPTY_BASES RC_<
	G_<
	NFeatureTag
	, TContext&
	, TActivation
	, TReactOrder
	HFSM2_IF_UTILITY_THEORY(, TRank, TUtility, TRNG)
	, NSubstitutionLimit
	HFSM2_IF_PLANS(, NTaskCapacity)
	, TPayload
	>
	, TApex
	>
	: public			RP_<
	G_<
	NFeatureTag
	, TContext&
	, TActivation
	, TReactOrder
	HFSM2_IF_UTILITY_THEORY(, TRank, TUtility, TRNG)
	, NSubstitutionLimit
	HFSM2_IF_PLANS(, NTaskCapacity)
	, TPayload
	>
	, TApex
	>
	{
	using Base =		RP_<
		G_<
		NFeatureTag
		, TContext&
		, TActivation
	, TReactOrder
	HFSM2_IF_UTILITY_THEORY(, TRank, TUtility, TRNG)
	, NSubstitutionLimit
	HFSM2_IF_PLANS(, NTaskCapacity)
	, TPayload
	>
	, TApex
	>;

	public:
	static constexpr FeatureTag FEATURE_TAG = Base::FEATURE_TAG;

	using typename Base::Context;

#if HFSM2_UTILITY_THEORY_AVAILABLE()
	using typename Base::RNG;
#endif

#if HFSM2_LOG_INTERFACE_AVAILABLE()
	using typename Base::Logger;
#endif

	public:
	using Base::Base;

	private:
	using Base::_core;
};

// TContext*

template <
	FeatureTag NFeatureTag
  , typename TContext
  , typename TActivation
  , typename TReactOrder

#if HFSM2_UTILITY_THEORY_AVAILABLE()
, typename TRank
, typename TUtility
  , typename TRNG
#endif

, Short NSubstitutionLimit
  HFSM2_IF_PLANS(, Long NTaskCapacity)
, typename TPayload
  , typename TApex
>
class HFSM2_EMPTY_BASES RC_<
							G_<
								NFeatureTag
							  , TContext*
							  , TActivation
							  , TReactOrder
							  HFSM2_IF_UTILITY_THEORY(, TRank, TUtility, TRNG)
							  , NSubstitutionLimit
							  HFSM2_IF_PLANS(, NTaskCapacity)
							  , TPayload
							>
						  , TApex
						>
	: public			RP_<
							G_<
								NFeatureTag
							  , TContext*
							  , TActivation
							  , TReactOrder
							  HFSM2_IF_UTILITY_THEORY(, TRank, TUtility, TRNG)
							  , NSubstitutionLimit
							  HFSM2_IF_PLANS(, NTaskCapacity)
							  , TPayload
							>
						  , TApex
						>
{
	using Base =		RP_<
	G_<
	NFeatureTag
	, TContext*
	, TActivation
							  , TReactOrder
							  HFSM2_IF_UTILITY_THEORY(, TRank, TUtility, TRNG)
							  , NSubstitutionLimit
							  HFSM2_IF_PLANS(, NTaskCapacity)
							  , TPayload
							>
						  , TApex
						>;

public:
static constexpr FeatureTag FEATURE_TAG = Base::FEATURE_TAG;

	using typename Base::Context;

#if HFSM2_UTILITY_THEORY_AVAILABLE()
	using typename Base::RNG;
#endif

#if HFSM2_LOG_INTERFACE_AVAILABLE()
	using typename Base::Logger;
#endif

public:
#if HFSM2_UTILITY_THEORY_AVAILABLE()

	HFSM2_CONSTEXPR(14)	explicit RC_(Context context
								   , RNG& rng
								   HFSM2_IF_LOG_INTERFACE(, Logger* const logger = nullptr))	noexcept;

#else

	HFSM2_CONSTEXPR(14)	explicit RC_(Context context = nullptr
								   HFSM2_IF_LOG_INTERFACE(, Logger* const logger = nullptr))	noexcept;

#endif

	HFSM2_CONSTEXPR(NO)	RC_(const RC_& )														noexcept = default;
	HFSM2_CONSTEXPR(NO)	RC_(	  RC_&&)														noexcept = default;

	HFSM2_CONSTEXPR(14)	void setContext(Context context)										noexcept	{ _core.context = context; }

private:
	using Base::_core;
};

// TContext == EmptyContext

template <
	FeatureTag NFeatureTag
  , typename TActivation
  , typename TReactOrder

#if HFSM2_UTILITY_THEORY_AVAILABLE()
, typename TRank
, typename TUtility
  , typename TRNG
#endif

, Short NSubstitutionLimit
  HFSM2_IF_PLANS(, Long NTaskCapacity)
, typename TPayload
  , typename TApex
>
class HFSM2_EMPTY_BASES RC_<
							G_<
								NFeatureTag
							  , EmptyContext
							  , TActivation
							  , TReactOrder
							  HFSM2_IF_UTILITY_THEORY(, TRank, TUtility, TRNG)
							  , NSubstitutionLimit
							  HFSM2_IF_PLANS(, NTaskCapacity)
							  , TPayload
							>
						  , TApex
						>
	: public			RP_<
							G_<
								NFeatureTag
							  , EmptyContext
							  , TActivation
							  , TReactOrder
							  HFSM2_IF_UTILITY_THEORY(, TRank, TUtility, TRNG)
							  , NSubstitutionLimit
							  HFSM2_IF_PLANS(, NTaskCapacity)
							  , TPayload
							>
						  , TApex
						>
	, public	 EmptyContext
{
	using Base =		RP_<
	G_<
	NFeatureTag
	, EmptyContext
	, TActivation
	, TReactOrder
							  HFSM2_IF_UTILITY_THEORY(, TRank, TUtility, TRNG)
							  , NSubstitutionLimit
							  HFSM2_IF_PLANS(, NTaskCapacity)
							  , TPayload
							>
						  , TApex
						>;

public:
static constexpr FeatureTag FEATURE_TAG = Base::FEATURE_TAG;

#if HFSM2_UTILITY_THEORY_AVAILABLE()
	using typename Base::RNG;
#endif

#if HFSM2_LOG_INTERFACE_AVAILABLE()
	using typename Base::Logger;
#endif

public:

#if HFSM2_UTILITY_THEORY_AVAILABLE()

	HFSM2_CONSTEXPR(14)	explicit RC_(RNG& rng
								   HFSM2_IF_LOG_INTERFACE(, Logger* const logger = nullptr))	noexcept;

#else

	HFSM2_CONSTEXPR(14)	explicit RC_(HFSM2_IF_LOG_INTERFACE(Logger* const logger = nullptr))	noexcept;

#endif

	HFSM2_CONSTEXPR(NO)	RC_(const RC_& )														noexcept = default;
	HFSM2_CONSTEXPR(NO)	RC_(	  RC_&&)														noexcept = default;
};

}
}

namespace hfsm2 {
	namespace detail {

		template <FeatureTag NFT_, typename TC_, typename TV_, typename TRO_ HFSM2_IF_UTILITY_THEORY(, typename TR_, typename TU_, typename TG_), Short NSL_ HFSM2_IF_PLANS(, Long NTC_), typename TP_, typename TA_>
		HFSM2_CONSTEXPR(14)
		RC_<G_<NFT_, TC_, TV_, TRO_ HFSM2_IF_UTILITY_THEORY(, TR_, TU_, TG_), NSL_ HFSM2_IF_PLANS(, NTC_), TP_>, TA_>::RC_(Context& context
		HFSM2_IF_UTILITY_THEORY(, RNG& rng)
		HFSM2_IF_LOG_INTERFACE(, Logger* const logger)) noexcept
		: Base{context
		HFSM2_IF_UTILITY_THEORY(, rng)
	HFSM2_IF_LOG_INTERFACE(, logger)}
{}

template <FeatureTag NFT_, typename TC_, typename TV_, typename TRO_ HFSM2_IF_UTILITY_THEORY(, typename TR_, typename TU_, typename TG_), Short NSL_ HFSM2_IF_PLANS(, Long NTC_), typename TP_, typename TA_>
HFSM2_CONSTEXPR(14)
RC_<G_<NFT_, TC_, TV_, TRO_ HFSM2_IF_UTILITY_THEORY(, TR_, TU_, TG_), NSL_ HFSM2_IF_PLANS(, NTC_), TP_>, TA_>::RC_(PureContext&& context
																												 HFSM2_IF_UTILITY_THEORY(, RNG& rng)
																												 HFSM2_IF_LOG_INTERFACE(, Logger* const logger)) noexcept
	: Base{move(context)
		 HFSM2_IF_UTILITY_THEORY(, rng)
		 HFSM2_IF_LOG_INTERFACE(, logger)}
{}

#if HFSM2_UTILITY_THEORY_AVAILABLE()

template <FeatureTag NFT_, typename TC_, typename TV_, typename TRO_, typename TR_, typename TU_, typename TG_, Short NSL_ HFSM2_IF_PLANS(, Long NTC_), typename TP_, typename TA_>
HFSM2_CONSTEXPR(14)
RC_<G_<NFT_, TC_*, TV_, TRO_, TR_, TU_, TG_, NSL_ HFSM2_IF_PLANS(, NTC_), TP_>, TA_>::RC_(Context context
																						, RNG& rng
																						HFSM2_IF_LOG_INTERFACE(, Logger* const logger)) noexcept
: Base{context
		 , rng
		 HFSM2_IF_LOG_INTERFACE(, logger)}
{}

#else

template <FeatureTag NFT_, typename TC_, typename TV_, typename TRO_, Short NSL_ HFSM2_IF_PLANS(, Long NTC_), typename TP_, typename TA_>
HFSM2_CONSTEXPR(14)
RC_<G_<NFT_, TC_*, TV_, TRO_, NSL_ HFSM2_IF_PLANS(, NTC_), TP_>, TA_>::RC_(Context context
																		 HFSM2_IF_LOG_INTERFACE(, Logger* const logger)) noexcept
	: Base{context
		 HFSM2_IF_LOG_INTERFACE(, logger)}
{}

#endif

#if HFSM2_UTILITY_THEORY_AVAILABLE()

template <FeatureTag NFT_, typename TV_, typename TRO_, typename TR_, typename TU_, typename TG_, Short NSL_ HFSM2_IF_PLANS(, Long NTC_), typename TP_, typename TA_>
HFSM2_CONSTEXPR(14)
RC_<G_<NFT_, EmptyContext, TV_, TRO_, TR_, TU_, TG_, NSL_ HFSM2_IF_PLANS(, NTC_), TP_>, TA_>::RC_(RNG& rng
																								HFSM2_IF_LOG_INTERFACE(, Logger* const logger)) noexcept
	: Base{static_cast<EmptyContext&>(*this)
		 , rng
		 HFSM2_IF_LOG_INTERFACE(, logger)}
{}

#else

template <FeatureTag NFT_, typename TV_, typename TRO_, Short NSL_ HFSM2_IF_PLANS(, Long NTC_), typename TP_, typename TA_>
HFSM2_CONSTEXPR(14)
RC_<G_<NFT_, EmptyContext, TV_, TRO_, NSL_ HFSM2_IF_PLANS(, NTC_), TP_>, TA_>::RC_(HFSM2_IF_LOG_INTERFACE(Logger* const logger)) noexcept
	: Base{static_cast<EmptyContext&>(*this)
		 HFSM2_IF_LOG_INTERFACE(, logger)}
{}

#endif

}
}

namespace hfsm2 {
	namespace detail {

		/// @brief FSM Root
		/// @tparam `TConfig` Type configuration
		/// @tparam `TApex` Root region type
		template <
		typename TConfig
		, typename TApex
		>
		class HFSM2_EMPTY_BASES InstanceT final
		: public	 RC_<TConfig, TApex>
		{
		using Base = RC_<TConfig, TApex>;

		public:
		using Base::Base;
	};

#if HFSM2_UTILITY_THEORY_AVAILABLE()

	// TRNG == RNGT<TUtility>

	/// @brief FSM Root
	/// @tparam `TConfig` Type configuration
	/// @tparam `TApex` Root region type
	template <
	FeatureTag NFeatureTag
	, typename TContext
	, typename TActivation
	, typename TReactOrder
	, typename TRank
	, typename TUtility
	, Short NSubstitutionLimit
	HFSM2_IF_PLANS(, Long NTaskCapacity)
	, typename TPayload
	, typename TApex
	>
	class HFSM2_EMPTY_BASES InstanceT<
		G_<
		NFeatureTag
		, TContext
		, TActivation
		, TReactOrder
		, TRank
		, TUtility
		, RNGT<TUtility>
		, NSubstitutionLimit
		HFSM2_IF_PLANS(, NTaskCapacity)
		, TPayload
		>
	, TApex
	> final
	: public			RC_<
		G_<
		NFeatureTag
		, TContext
		, TActivation
		, TReactOrder
		, TRank
		, TUtility
		, RNGT<TUtility>
		, NSubstitutionLimit
		HFSM2_IF_PLANS(, NTaskCapacity)
		, TPayload
		>
	, TApex
	>
	, public			RNGT<TUtility>
	{
	using Base =		RC_<
		G_<
		NFeatureTag
		, TContext
		, TActivation
		, TReactOrder
		, TRank
		, TUtility
		, RNGT<TUtility>
		, NSubstitutionLimit
	HFSM2_IF_PLANS(, NTaskCapacity)
	, TPayload
	>
	, TApex
	>;

	public:
	static constexpr FeatureTag FEATURE_TAG = Base::FEATURE_TAG;

	using typename Base::Context;

#if HFSM2_LOG_INTERFACE_AVAILABLE()
	using typename Base::Logger;
#endif

	public:
	HFSM2_CONSTEXPR(14)	explicit InstanceT(Context& context
	HFSM2_IF_LOG_INTERFACE(, Logger* const logger = nullptr))	noexcept
	: Base{context
	, static_cast<RNGT<TUtility>&>(*this)
HFSM2_IF_LOG_INTERFACE(, logger)}
		, RNGT<TUtility>{0}
	{}
};

// TContext == EmptyContext
// TRNG == RNGT<TUtility>

/// @brief FSM Root
/// @tparam `TConfig` Type configuration
/// @tparam `TApex` Root region type
template <
	FeatureTag NFeatureTag
  , typename TActivation
  , typename TReactOrder
  , typename TRank
  , typename TUtility
  , Short NSubstitutionLimit
  HFSM2_IF_PLANS(, Long NTaskCapacity)
  , typename TPayload
  , typename TApex
>
class HFSM2_EMPTY_BASES InstanceT<
	G_<
	NFeatureTag
	, EmptyContext
	, TActivation
	, TReactOrder
	, TRank
	, TUtility
	, RNGT<TUtility>
	, NSubstitutionLimit
	HFSM2_IF_PLANS(, NTaskCapacity)
	, TPayload
	>
						  , TApex
						> final
: public			RC_<
	G_<
	NFeatureTag
	, EmptyContext
	, TActivation
	, TReactOrder
	, TRank
	, TUtility
	, RNGT<TUtility>
	, NSubstitutionLimit
	HFSM2_IF_PLANS(, NTaskCapacity)
	, TPayload
	>
						  , TApex
						>
	, public RNGT<TUtility>
{
	using Base =		RC_<
	G_<
	NFeatureTag
	, EmptyContext
	, TActivation
	, TReactOrder
	, TRank
	, TUtility
	, RNGT<TUtility>
	, NSubstitutionLimit
							  HFSM2_IF_PLANS(, NTaskCapacity)
							  , TPayload
							>
						  , TApex
						>;

public:
static constexpr FeatureTag FEATURE_TAG = Base::FEATURE_TAG;

#if HFSM2_LOG_INTERFACE_AVAILABLE()
	using typename Base::Logger;
#endif

public:
	HFSM2_CONSTEXPR(14)	explicit InstanceT(HFSM2_IF_LOG_INTERFACE(Logger* const logger = nullptr))	noexcept
		: Base{static_cast<RNGT<TUtility>&>(*this)
			 HFSM2_IF_LOG_INTERFACE(, logger)}
		, RNGT<TUtility>{0}
	{}
};

#endif

}
}

#if defined(__GNUC__) || defined(__GNUG__)
#pragma GCC diagnostic pop
#endif

#ifdef __clang__
#pragma clang diagnostic pop
#endif

#if _MSC_VER == 1900
#pragma warning(pop)
#endif

#undef HFSM2_UNUSED

#undef HFSM2_ATTRIBUTE

#undef HFSM2_ATTRIBUTE_FALLTHROUGH

#undef HFSM2_ATTRIBUTE_NO_UNIQUE_ADDRESS

#undef HFSM2_CONSTEXPR

#undef HFSM2_CONSTEXPR_NO

#undef HFSM2_CONSTEXPR_11

#undef HFSM2_CONSTEXPR_14

#undef HFSM2_CONSTEXPR_17

#undef HFSM2_CONSTEXPR_20

//#undef HFSM2_EMPTY_BASES

//#undef HFSM2_ARCHITECTURE
//#undef HFSM2_ARCHITECTURE_64
//#undef HFSM2_ARCHITECTURE_32
#undef HFSM2_64BIT_OR_32BIT

//#undef HFSM2_BREAK
#undef HFSM2_BREAK_AVAILABLE

#undef HFSM2_IF_DEBUG
#undef HFSM2_UNLESS_DEBUG
#undef HFSM2_DEBUG_OR

//#undef HFSM2_ASSERT_AVAILABLE
#undef HFSM2_IF_ASSERT
//#undef HFSM2_CHECKED
#undef HFSM2_ASSERT
#undef HFSM2_ASSERT_OR

#undef HFSM2_EXPLICIT_MEMBER_SPECIALIZATION_AVAILABLE

#undef HFSM2_IF_TYPEINDEX
#undef HFSM2_TYPEINDEX_AVAILABLE
#undef HFSM2_IF_TYPEINDEX

//#undef HFSM2_DEBUG_STATE_TYPE_AVAILABLE

#undef HFSM2_PLANS_AVAILABLE
#undef HFSM2_IF_PLANS

#undef HFSM2_SERIALIZATION_AVAILABLE
#undef HFSM2_IF_SERIALIZATION

#undef HFSM2_STRUCTURE_REPORT_AVAILABLE
#undef HFSM2_IF_STRUCTURE_REPORT

#undef HFSM2_TRANSITION_HISTORY_AVAILABLE
#undef HFSM2_IF_TRANSITION_HISTORY

#undef HFSM2_UTILITY_THEORY_AVAILABLE
#undef HFSM2_IF_UTILITY_THEORY

#undef HFSM2_VERBOSE_DEBUG_LOG_AVAILABLE

#undef HFSM2_LOG_INTERFACE_AVAILABLE
#undef HFSM2_IF_LOG_INTERFACE

#undef HFSM2_LOG_TRANSITION

#ifdef HFSM2_ENABLE_PLANS
#undef HFSM2_LOG_TASK_STATUS
#undef HFSM2_LOG_PLAN_STATUS
#endif

#undef HFSM2_LOG_CANCELLED_PENDING

#ifdef HFSM2_UTILITY_THEORY_AVAILABLE
#undef HFSM2_LOG_UTILITY_RESOLUTION
#undef HFSM2_LOG_RANDOM_RESOLUTION
#endif

#undef HFSM2_LOG_STATE_METHOD
```

#### States.hpp
```cpp
//==============================================================================
//
// Title:		States Definitions and transitions for traffic light
//
// Created on:	8/29/2025 at 11:18:29 AM by AD.
//
//==============================================================================
#include "machine.hpp"

// data shared between FSM states and outside code
struct Context {
	unsigned cycleCount = 0;
	unsigned countGreenBlinking = 0;
	unsigned countGreen = 0;
	unsigned countYellow = 0;
	unsigned countRed = 0;
};

// convenience typedef
using M = hfsm2::MachineT<hfsm2::Config::ContextT<Context>>;

// macro magic invoked to simplify FSM structure declaration
#define S(s) struct s

// State machine structure
using FSM = M::PeerRoot<
	// sub-machine ..
	M::Composite<S(On),
	// .. with 5 sub-states
	S(Red),
	S(YellowDownwards),
	S(YellowUpwards),
	S(GreenBlinking),
	S(Green)
	>,
				S(Off)
			>;
#undef S

//------------------------------------------------------------------------------

static_assert(FSM::regionId<On>()			  ==  1, "");

static_assert(FSM::stateId<On>()			  ==  1, "");
static_assert(FSM::stateId<Red>()			  ==  2, "");
static_assert(FSM::stateId<YellowDownwards>() ==  3, "");
static_assert(FSM::stateId<YellowUpwards>()	  ==  4, "");
static_assert(FSM::stateId<GreenBlinking>()	  ==  5, "");
static_assert(FSM::stateId<Green>()			  ==  6, "");
static_assert(FSM::stateId<Off>()			  ==  7, "");

////////////////////////////////////////////////////////////////////////////////

// top-level region in the hierarchy
struct On
	: FSM::State // necessary boilerplate!
{
	// called on state entry
	void enter(Control& control) {
		control.context().cycleCount = 0;
		TraceMessage("On");
	}
};

//------------------------------------------------------------------------------

// sub-states
struct Red
	: FSM::State
{
	void enter(Control& control) {
		++control.context().cycleCount;
		LightRed = true;
		LightYellow = false;
		LightGreen = false;
		control.context().countRed = 0;
		CountDown = DurationRed + DurationYellow + 2;
		TraceMessage("Red");

	}

	// state can initiate transitions to _any_ other state
	void update(FullControl& control) {
		if (control.context().countRed++ >= DurationRed){
			control.changeTo<YellowDownwards>();
		}
	CountDown--;
	}
};

// - - - - - - - - - - - - - - - - - - - - - - - - - - - - - - - - - - - - - - -

struct YellowDownwards
	: FSM::State
{
	void enter(Control& control) {
		TraceMessage("Yellow v");
		LightYellow = true; //Keep Red On
		control.context().countYellow = 0;
	}

	void update(FullControl& control) {
		if (control.context().countYellow++ > DurationYellow) { //was 3
			control.changeTo<Green>();
		}
		CountDown--;
	}
};

// - - - - - - - - - - - - - - - - - - - - - - - - - - - - - - - - - - - - - - -

struct YellowUpwards
	: FSM::State
{
	void enter(Control& control) {
		TraceMessage("Yellow ^");
		LightGreen = false;
		LightYellow = true;
		CountDownGreenON = false;
		control.context().countYellow = 0;
	}

	void update(FullControl& control) {
		if (control.context().countYellow++ > DurationYellow) {
			control.changeTo<Red>();
		}
	}
};

// - - - - - - - - - - - - - - - - - - - - - - - - - - - - - - - - - - - - - - -

struct GreenBlinking
	: FSM::State
{
	void enter(Control& control) {
		TraceMessage("Green Blinking");
		CountDownGreenON = true;
		control.context().countGreenBlinking = 0;
	}

	void update(FullControl& control) {
		LightGreen = !LightGreen; // Blinking
		if ((control.context().countGreenBlinking++ > DurationGreenBlinking) && !LightGreen) {
			control.changeTo<YellowUpwards>();
		}
		CountDown--;
	}
};

// - - - - - - - - - - - - - - - - - - - - - - - - - - - - - - - - - - - - - - -

struct Green
	: FSM::State
{
	void enter(Control& control) {
		TraceMessage("Green");
		control.context().countGreen = 0;
		LightRed = false;
		LightYellow = false;
		LightGreen = true;
		CountDownGreenON = true;
		CountDown = DurationGreen + DurationGreenBlinking + 4;
	}

	void update(FullControl& control) {
		if (control.context().countGreen++ > DurationGreen){
			control.changeTo<GreenBlinking>();
		}
		CountDown--;
	}
};

//------------------------------------------------------------------------------

// another top-level state
struct Off
	: FSM::State
{
	void enter(Control&) {
		TraceMessage("Off");
	}
};
```

- Visualisation Logical/mappView (not shown)

Listed in the project but not available here: Logical/Global.typ, Logical/Global.var, Logical/Libraries, Logical/Ampel/Types.typ, Logical/Ampel/Logging.hpp
